FUNCTION_BLOCK FB_CrectCamYaDaoUpDown2	
VAR_INPUT
   	bCreatTable		                         :BOOL;	
	Reset                                        :BOOL;  
	iTable		                                :UINT;    

    fMoveLength                              :REAL:=8;   //升降最大距离
    fSaveLength1                               :REAL:=2 ;    //压针抬升高度
    fSaveLength2                               :REAL:=3;  //压针下压高度

    fMasterKeyPos1                           :REAL:=144;   
    fMasterKeyPos2                           :REAL:=164;   
    fMasterKeyPos3                           :REAL:=204;   

    fMasterKeyPos4                           :REAL:=246;   
    fMasterKeyPos5                          :REAL:=289;   
    fMasterKeyPos6                           :REAL:=328;   


END_VAR

VAR_IN_OUT
	axisSlave		                            :axis_ref;  
	axisMaster		                            :axis_ref;  
END_VAR

VAR_OUTPUT
    bCreatTableDone                        :BOOL;
    bCreatTableError                        :BOOL;
	bError                         :BOOL;

END_VAR


VAR
	rtrigs		                                      :ARRAY[1..3]OF R_TRIG;
	ftrigs		                                      :ARRAY[1..3]OF F_TRIG;
    PositionData1			                  :ARRAY[1..8] OF MC_MotionFunctionPoint;	////
	fbCamtableselect:		               	MC_CamTableSelect;////
	Cam_table:				MC_CAM_REF;////
	bWriteCamData: BOOL;
    iCreatTableStep       :INT;
END_VAR


rtrigs[1](CLK:=bCreatTable);  
ftrigs[1](CLK:=bCreatTable);  

CASE iCreatTableStep OF   
0:  
    IF  rtrigs[1].Q  AND NOT bCreatTableError  THEN
         fbCamtableselect.Execute:=FALSE;
         bCreatTableDone:=FALSE;
         bCreatTable:=FALSE;
         bWriteCamData:=TRUE;
         iCreatTableStep:=10;
    END_IF 

10: 
   IF NOT bWriteCamData THEN 
	  fbCamtableselect.Execute:=TRUE;   
	 iCreatTableStep:=20;	
  END_IF

20:		
	IF NOT  fbCamtableselect.Execute   THEN
        bCreatTableDone:=TRUE;
		iCreatTableStep:=0;	
    ELSIF  fbCamtableselect.Error        THEN
       bCreatTableError:=TRUE;
       iCreatTableStep:=999;	//创建凸轮失败
	END_IF		
END_CASE

(**********故障***********)
	IF  Reset  AND bCreatTableError  THEN  
	   bCreatTableError:=FALSE;
	   iCreatTableStep:=0;
	END_IF


ModifyCam();

ACTION ModifyCam:

fbCamtableselect(   
	Execute:=                        fbCamtableselect.Execute ,
	Periodic:=                        FALSE ,
	MasterAbsolute:=             FALSE,
	SlaveAbsolute:=                FALSE ,
	CamTableID:=                  iTable,
	Master:=                         axisMaster ,
	Slave:=                            axisSlave ,
	CamTable:=                     Cam_table , );

IF fbCamtableselect.Done THEN
    fbCamtableselect.Execute:=FALSE;
END_IF

IF bWriteCamData  THEN
 
	  Cam_table.ArraySize:=SIZEOF(PositionData1); 
	  Cam_table.NoOfColumns:=1;
	  Cam_table.NoOfRows:=7;
	  Cam_table.pArray:=ADR(PositionData1);
	  Cam_table.TableType:=MC_TABLETYPE_MOTIONFUNCTION;
      //MOTIONFUNCTYPE_BESCHLTRAPEZ     MOTIONFUNCTYPE_POLYNOM7_MM    MOTIONFUNCTYPE_BESCHLTRAPEZ   MOTIONFUNCTYPE_POLYNOM1

	  PositionData1[1].	PointIndex	:=	        1;
	  PositionData1[1].	FunctionType	:=		MOTIONFUNCTYPE_POLYNOM1;//
	  PositionData1[1].	PointType	:=	        MOTIONPOINTTYPE_MOTION;
	  PositionData1[1].	RelIndexNextPoint	:=  1;
	  PositionData1[1].	MasterPos	:=	        0;
	  PositionData1[1].	SlavePos	:=	        0;		//fMoveLength
	  PositionData1[1].	SlaveVelo	:=	        0;
	  
	  PositionData1[2].	PointIndex	:=	        2;
	  PositionData1[2].	FunctionType	:=		MOTIONFUNCTYPE_POLYNOM5_MM;
	  PositionData1[2].	PointType	:=	        MOTIONPOINTTYPE_MOTION;
	  PositionData1[2].	RelIndexNextPoint	:=  1;
	  PositionData1[2].	MasterPos	:=	        fMasterKeyPos1;
	  PositionData1[2].	SlavePos	:=	        0;	
	  PositionData1[2].	SlaveVelo	:=	       0	;

	  PositionData1[3].	PointIndex	:=	        3;
	  PositionData1[3].	FunctionType	:=		MOTIONFUNCTYPE_POLYNOM1;
	  PositionData1[3].	PointType	:=	        MOTIONPOINTTYPE_MOTION;
	  PositionData1[3].	RelIndexNextPoint	:=  0;
	  PositionData1[3].	MasterPos	:=	        fMasterKeyPos2;
	  PositionData1[3].	SlavePos	:=	        fSaveLength1;	
	  PositionData1[3].	SlaveVelo	:=	        0	;

	  PositionData1[4].	PointIndex	:=	        4;
	  PositionData1[4].	FunctionType	:=		MOTIONFUNCTYPE_POLYNOM5_MM;
	  PositionData1[4].	PointType	:=	        MOTIONPOINTTYPE_MOTION;
	  PositionData1[4].	RelIndexNextPoint	:=  1;
	  PositionData1[4].	MasterPos	:=	        fMasterKeyPos3;
	  PositionData1[4].	SlavePos	:=	        fSaveLength1;	
	  PositionData1[4].	SlaveVelo	:=	       0	;

	  PositionData1[5].	PointIndex	:=	        5;
	  PositionData1[5].	FunctionType	:=		MOTIONFUNCTYPE_POLYNOM5_MM;
	  PositionData1[5].	PointType	:=	        MOTIONPOINTTYPE_MOTION;
	  PositionData1[5].	RelIndexNextPoint	:=  1;
	  PositionData1[5].	MasterPos	:=	        fMasterKeyPos4;
	  PositionData1[5].	SlavePos	:=	        fMoveLength;	
	  PositionData1[5].	SlaveVelo	:=	       0	;
(*
	  PositionData1[6].	PointIndex	:=	        6;
	  PositionData1[6].	FunctionType	:=		MOTIONFUNCTYPE_POLYNOM7_MM;
	  PositionData1[6].	PointType	:=	        MOTIONPOINTTYPE_MOTION;
	  PositionData1[6].	RelIndexNextPoint	:=  1;
	  PositionData1[6].	MasterPos	:=	        fMasterKeyPos5;
	  PositionData1[6].	SlavePos	:=	       fSaveLength2 ;	
	  PositionData1[6].	SlaveVelo	:=	        (fSaveLength2-fMoveLength)/ (fMasterKeyPos5-fMasterKeyPos4 )	;
*)
	  PositionData1[6].	PointIndex	:=	        6;
	  PositionData1[6].	FunctionType	:=		MOTIONFUNCTYPE_POLYNOM1;
	  PositionData1[6].	PointType	:=	        MOTIONPOINTTYPE_MOTION;
	  PositionData1[6].	RelIndexNextPoint	:=  1;
	  PositionData1[6].	MasterPos	:=	        fMasterKeyPos6;
	  PositionData1[6].	SlavePos	:=	        fSaveLength2;	
	  PositionData1[6].	SlaveVelo	:=	        0	;

	  PositionData1[7].	PointIndex	:=	        7;
	  PositionData1[7].	FunctionType	:=		MOTIONFUNCTYPE_POLYNOM1;
	  PositionData1[7].	PointType	:=	        MOTIONPOINTTYPE_MOTION;
	  PositionData1[7].	RelIndexNextPoint	:=  0;
	  PositionData1[7].	MasterPos	:=	        360;
	  PositionData1[7].	SlavePos	:=	        fSaveLength2;	
	  PositionData1[7].	SlaveVelo	:=	        0	;

     bWriteCamData:=FALSE;
END_IF







(*

IF bWriteCamData  THEN
 
	  Cam_table.ArraySize:=SIZEOF(PositionData1); 
	  Cam_table.NoOfColumns:=1;
	  Cam_table.NoOfRows:=7;
	  Cam_table.pArray:=ADR(PositionData1);
	  Cam_table.TableType:=MC_TABLETYPE_MOTIONFUNCTION;
      //MOTIONFUNCTYPE_BESCHLTRAPEZ     MOTIONFUNCTYPE_POLYNOM7_MM    MOTIONFUNCTYPE_BESCHLTRAPEZ   MOTIONFUNCTYPE_POLYNOM1

	  PositionData1[1].	PointIndex	:=	        1;
	  PositionData1[1].	FunctionType	:=		MOTIONFUNCTYPE_POLYNOM1;//
	  PositionData1[1].	PointType	:=	        MOTIONPOINTTYPE_MOTION;
	  PositionData1[1].	RelIndexNextPoint	:=  1;
	  PositionData1[1].	MasterPos	:=	        0;
	  PositionData1[1].	SlavePos	:=	        0;		//fMoveLength
	  PositionData1[1].	SlaveVelo	:=	        0;
	  
	  PositionData1[2].	PointIndex	:=	        2;
	  PositionData1[2].	FunctionType	:=		MOTIONFUNCTYPE_POLYNOM5_MM;
	  PositionData1[2].	PointType	:=	        MOTIONPOINTTYPE_MOTION;
	  PositionData1[2].	RelIndexNextPoint	:=  1;
	  PositionData1[2].	MasterPos	:=	        fMasterKeyPos1;
	  PositionData1[2].	SlavePos	:=	        0;	
	  PositionData1[2].	SlaveVelo	:=	       0	;

	  PositionData1[3].	PointIndex	:=	        3;
	  PositionData1[3].	FunctionType	:=		MOTIONFUNCTYPE_POLYNOM1;
	  PositionData1[3].	PointType	:=	        MOTIONPOINTTYPE_MOTION;
	  PositionData1[3].	RelIndexNextPoint	:=  0;
	  PositionData1[3].	MasterPos	:=	        fMasterKeyPos2;
	  PositionData1[3].	SlavePos	:=	        fSaveLength1;	
	  PositionData1[3].	SlaveVelo	:=	        0	;

	  PositionData1[4].	PointIndex	:=	        4;
	  PositionData1[4].	FunctionType	:=		MOTIONFUNCTYPE_POLYNOM5_MM;
	  PositionData1[4].	PointType	:=	        MOTIONPOINTTYPE_MOTION;
	  PositionData1[4].	RelIndexNextPoint	:=  1;
	  PositionData1[4].	MasterPos	:=	        fMasterKeyPos3;
	  PositionData1[4].	SlavePos	:=	        fSaveLength1;	
	  PositionData1[4].	SlaveVelo	:=	       0	;

	  PositionData1[5].	PointIndex	:=	        5;
	  PositionData1[5].	FunctionType	:=		MOTIONFUNCTYPE_POLYNOM5_MM;
	  PositionData1[5].	PointType	:=	        MOTIONPOINTTYPE_MOTION;
	  PositionData1[5].	RelIndexNextPoint	:=  1;
	  PositionData1[5].	MasterPos	:=	        fMasterKeyPos4;
	  PositionData1[5].	SlavePos	:=	        fMoveLength;	
	  PositionData1[5].	SlaveVelo	:=	       0	;
(*
	  PositionData1[6].	PointIndex	:=	        6;
	  PositionData1[6].	FunctionType	:=		MOTIONFUNCTYPE_POLYNOM7_MM;
	  PositionData1[6].	PointType	:=	        MOTIONPOINTTYPE_MOTION;
	  PositionData1[6].	RelIndexNextPoint	:=  1;
	  PositionData1[6].	MasterPos	:=	        fMasterKeyPos5;
	  PositionData1[6].	SlavePos	:=	       fSaveLength2 ;	
	  PositionData1[6].	SlaveVelo	:=	        (fSaveLength2-fMoveLength)/ (fMasterKeyPos5-fMasterKeyPos4 )	;
*)
	  PositionData1[6].	PointIndex	:=	        6;
	  PositionData1[6].	FunctionType	:=		MOTIONFUNCTYPE_POLYNOM1;
	  PositionData1[6].	PointType	:=	        MOTIONPOINTTYPE_MOTION;
	  PositionData1[6].	RelIndexNextPoint	:=  1;
	  PositionData1[6].	MasterPos	:=	        fMasterKeyPos6;
	  PositionData1[6].	SlavePos	:=	        0;	
	  PositionData1[6].	SlaveVelo	:=	        0	;

	  PositionData1[7].	PointIndex	:=	        7;
	  PositionData1[7].	FunctionType	:=		MOTIONFUNCTYPE_POLYNOM1;
	  PositionData1[7].	PointType	:=	        MOTIONPOINTTYPE_MOTION;
	  PositionData1[7].	RelIndexNextPoint	:=  0;
	  PositionData1[7].	MasterPos	:=	        360;
	  PositionData1[7].	SlavePos	:=	        0;	
	  PositionData1[7].	SlaveVelo	:=	        0	;

     bWriteCamData:=FALSE;
END_IF

*)
END_ACTION

END_FUNCTION_BLOCK

(* stored: Version 1.1.0.1, ProductVersion 3.1.4024.12
   POU FB_CrectCamYaDaoUpDown2: Id {2a095bad-5aeb-4bef-bcc5-f4b33ee4d68c}, SpecialFunc None
   Action ModifyCam: Id {4f4cb7ad-d627-40f3-acfc-3658b64bafd8} *)
